// TIA Portal V17 export
// export: Created 2023-12-22T15:08:09.5884674Z, ExportSetting WithDefaults, DisplayName Totally Integrated Automation Portal, DisplayVersion V17, DisplayName TIA Portal Openness, DisplayVersion V17, DisplayName TIA Portal Version Control Interface, DisplayVersion V17, DisplayName STEP 7 Professional, DisplayVersion V17, DisplayName STEP 7 Safety, DisplayVersion V17, DisplayName WinCC Advanced, DisplayVersion V17
DATA_BLOCK "PS_Any_DB"   // DB20
VERSION : 0.1
// stored: AutoNumber false, DBAccessibleFromOPCUA true, DBAccessibleFromWebserver true, InstanceOfName PS_Any, InstanceOfType FB
"PS_Any"
   // VAR
   //    x : Array[0..10] of Real;
   //    Delta_PE : Real;
   //    Delta_LE_in : Real;
   //    Delta_LE_out : Real;
   // END_VAR
BEGIN
END_DATA_BLOCK
